// TIA Portal project "Urban Intersection Control System" (V17)

(* hardware
DEVICE "S7-1500/ET200MP station_1"  S7-1500 station
   slot 0: "Rail_0"  Rack  6ES7 590-1***0-0AA0
   slot 1: "PLC_UICS_01"  CPU 1512C-1 PN  6ES7 512-1CK00-0AB0  V2.9
      slot 3: "CPU display_1"  6ES7591-1AA00-0AA0
      slot 32768: "PROFINET interface_1"  X1
         slot 32769: "Port_1"  X1 P1
         slot 32770: "Port_2"  X1 P2
      slot 34817: "Virtual CP interface port_1"  Virtual CP interface port  Virtual CP interface port
*)

// ===== PLC "PLC_UICS_01"  CPU 1512C-1 PN =====

VAR_GLOBAL   // PLC tag table "UICS_Table"
   "PB_Ped_Main" AT %I10.2 : Bool;   // Push button for pedestrian crossing on Main Street
   "PB_Ped_Cross" AT %I10.3 : Bool;   // Push button for pedestrian crossing on Cross Street
   "EM_Main_Override" AT %I10.4 : Bool;   // Emergency override signal (e.g. ambulances) on Main Street
   "EM_Cross_Override" AT %I10.5 : Bool;   // Emergency override signal on Cross Street
   "SENSOR_Main_Vehicle" AT %I10.6 : Bool;   // Vehicle detection sensor on Main Street
   "SENSOR_Cross_Vehicle" AT %I10.7 : Bool;   // Vehicle detection sensor on Cross Street
   "TL_Main_Red" AT %Q4.0 : Bool;   // Red traffic light signal for Main Street
   "TL_Main_Yellow" AT %Q4.1 : Bool;   // Yellow traffic light signal for Main Street
   "TL_Main_Green" AT %Q4.2 : Bool;   // Green traffic light signal for Main Street
   "TL_Cross_Red" AT %Q4.3 : Bool;   // Red traffic light signal for Cross Street
   "TL_Cross_Yellow" AT %Q4.4 : Bool;   // Yellow traffic light signal for Cross Street
   "TL_Cross_Green" AT %Q4.5 : Bool;   // Green traffic light signal for Cross Street
   "PED_Main_Walk" AT %Q4.6 : Bool;   // Pedestrian walk signal for Main Street
   "PED_Main_Dontwalk" AT %Q4.7 : Bool;   // Pedestrian don’t-walk signal for Main Street
   "PED_Cross_Walk" AT %Q5.0 : Bool;   // Pedestrian walk signal for Cross Street
   "PED_Cross_DontWalk" AT %Q5.1 : Bool;   // Pedestrian don’t-walk signal for Cross Street
   "PED_Warning_Buzzer" AT %Q5.2 : Bool;   // Audible alert for pedestrian crossing
   "SYS_Stop" AT %I10.1 : Bool;   // Emergency stop function
   "SYS_Start" AT %I10.0 : Bool;   // Begins the system
END_VAR

DATA_BLOCK "Main_Control_System_DB"   // DB1
{ S7_Optimized_Access := 'TRUE' }
VERSION : 0.1
// stored: InstanceOfName Main_Control_System
"Main_Control_System"
BEGIN
END_DATA_BLOCK

// folder: System blocks/Program resources

DATA_BLOCK "Traffic_Timer_DB"   // DB2
{ S7_Optimized_Access := 'TRUE' }
AUTHOR : Simatic
FAMILY : IEC
NAME : IEC_TMR
VERSION : 1.0
// stored: InstanceOfName IEC_TIMER
"IEC_TIMER"
BEGIN
END_DATA_BLOCK

// folder: (top level)

FUNCTION_BLOCK "Main_Control_System"   // FB1, LAD
{ S7_Optimized_Access := 'TRUE' }
VERSION : 0.1
   VAR
      Timer_Activated : Bool;
      Started : Bool;
      System_Running : Bool;   // System is actively running
      Emergency_Stop : Bool;   // Emergency stop activated flag
      Traffic_Timer : TON_TIME;
   END_VAR
BEGIN

REGION Network 1: System Start
   // Starts the system if all conditions are met
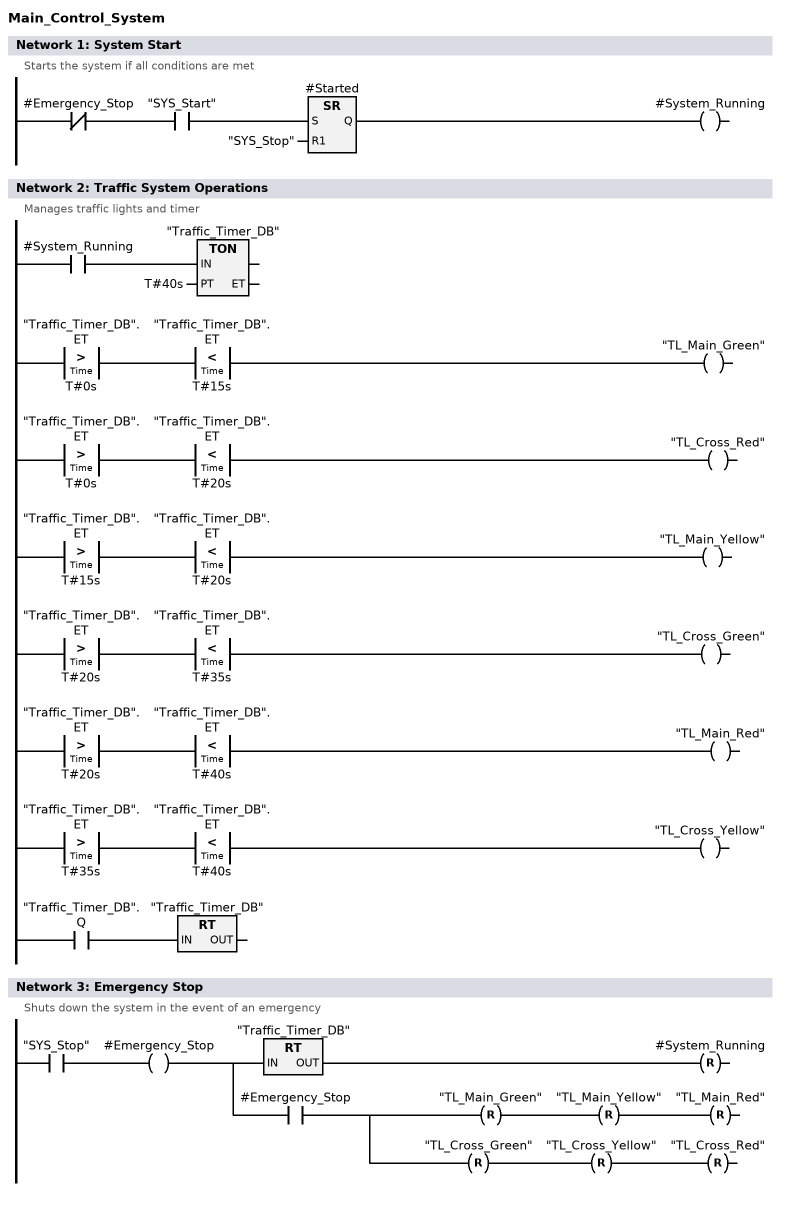
   RUNG wire#powerrail
      I_Contact( #Emergency_Stop )
      Contact( "SYS_Start" )
      S_SR(operand := #Started, r1 := "SYS_Stop")
      Coil( #System_Running )
   END_RUNG
   // the same network as SCL:
   IF NOT #Emergency_Stop AND "SYS_Start" THEN
       #Started := TRUE;   // SR flip-flop
   END_IF;
   IF "SYS_Stop" THEN #Started := FALSE; END_IF;
   #System_Running := #Started;
END_REGION

REGION Network 2: Traffic System Operations
   // Manages traffic lights and timer
   "Traffic_Timer_DB".TON(IN := #System_Running, PT := T#40s);
   "TL_Main_Green" := ("Traffic_Timer_DB".ET > T#0s) AND ("Traffic_Timer_DB".ET < T#15s);
   "TL_Cross_Red" := ("Traffic_Timer_DB".ET > T#0s) AND ("Traffic_Timer_DB".ET < T#20s);
   "TL_Main_Yellow" := ("Traffic_Timer_DB".ET > T#15s) AND ("Traffic_Timer_DB".ET < T#20s);
   "TL_Cross_Green" := ("Traffic_Timer_DB".ET > T#20s) AND ("Traffic_Timer_DB".ET < T#35s);
   "TL_Main_Red" := ("Traffic_Timer_DB".ET > T#20s) AND ("Traffic_Timer_DB".ET < T#40s);
   "TL_Cross_Yellow" := ("Traffic_Timer_DB".ET > T#35s) AND ("Traffic_Timer_DB".ET < T#40s);
   IF "Traffic_Timer_DB".Q THEN RESET_TIMER("Traffic_Timer_DB"); END_IF;
END_REGION

REGION Network 3: Emergency Stop
   // Shuts down the system in the event of an emergency
   RUNG wire#powerrail
      Contact( "SYS_Stop" )
      Coil( #Emergency_Stop )
      wire#w1
      RT_Coil( "Traffic_Timer_DB" )
      R_Coil( #System_Running )
   END_RUNG
   RUNG wire#w1
      Contact( #Emergency_Stop )
      wire#w2
      R_Coil( "TL_Main_Green" )
      R_Coil( "TL_Main_Yellow" )
      R_Coil( "TL_Main_Red" )
   END_RUNG
   RUNG wire#w2
      R_Coil( "TL_Cross_Green" )
      R_Coil( "TL_Cross_Yellow" )
      R_Coil( "TL_Cross_Red" )
   END_RUNG
   // the same network as SCL:
   #Emergency_Stop := "SYS_Stop";
   IF "SYS_Stop" THEN
       RESET_TIMER("Traffic_Timer_DB");
       #System_Running := FALSE;
   END_IF;
   IF "SYS_Stop" AND #Emergency_Stop THEN
       "TL_Main_Green" := FALSE;
       "TL_Main_Yellow" := FALSE;
       "TL_Main_Red" := FALSE;
       "TL_Cross_Green" := FALSE;
       "TL_Cross_Yellow" := FALSE;
       "TL_Cross_Red" := FALSE;
   END_IF;
END_REGION
END_FUNCTION_BLOCK

ORGANIZATION_BLOCK "Main"   // OB1, LAD, ProgramCycle
TITLE = "Main Program Sweep (Cycle)"
{ S7_Optimized_Access := 'TRUE' }
VERSION : 0.1
   VAR_INPUT
      Initial_Call : Bool;   // Initial call of this OB
      Remanence : Bool;   // =True, if remanent data are available
   END_VAR
BEGIN

REGION Network 1: Main
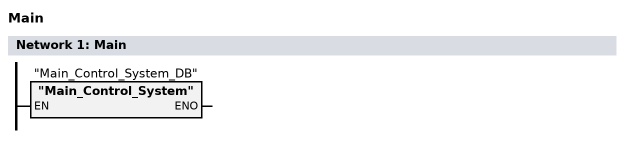
   RUNG wire#powerrail
      "Main_Control_System_DB"()
   END_RUNG
   // the same network as SCL:
   "Main_Control_System_DB"();   // "Main_Control_System"
END_REGION
END_ORGANIZATION_BLOCK